PROGRAM PRG_ReadModbusSensorData
VAR
	
	CurrentReadTarget			: EN_ModbusReadTarget := EN_ModbusReadTarget.READ_TARGET_PH;
	
	ProcessValueRegister		: WORD := 2089;
	TemperatureRegister			: WORD := 2409;
	PhSensorUnitId				: BYTE := 1;
	OrpSensorUnitId				: BYTE := 2;
	RegQuantityToRead			: WORD :=10;
	
	currentUnitId				: BYTE := PhSensorUnitId;
	currentModbusRegister		: WORD := ProcessValueRegister;

	ModbusBusy					: BOOL := FALSE;

	(* diagnostics *)	
	LastModbusError				: ST_ModbusErrorDiagnostics;
	LastErrorstate				: INT;
	CurrentState				: INT;
	CounterError				: INT := 0;
	CounterSuccess				: INT := 0;
	
	firstCall					: BOOL := TRUE;	
	
	scaleFactorPh				: REAL :=   1.219512195; (* 0.980167935 *);  		
	offsetPh					: REAL := 	-1.280487805; (* -0.0216290391086993 *);	


	scaleFactorOrp				: REAL := 0.999321727334388;
	offsetOrp					: REAL := 0.0;			
	
END_VAR

(* looping through pH, pH-T, ORP, ORP-T reading the latest values *)
IF firstCall THEN
	PhModbus.ReadRegs( Execute := FALSE);
	OrpModbus.ReadRegs( Execute := FALSE);
	firstCall := FALSE;
END_IF	

CASE  CurrentReadTarget OF 
	EN_ModbusReadTarget.READ_TARGET_PH:
		PhModbus.Readregs (UnitID 		:= PhSensorUnitId ,
   							Quantity   	:= RegQuantityToRead,
   							MBAddr    	:= ProcessValueRegister,
   							cbLength    := RegQuantityToRead*2,
   							pMemoryAddr := ADR(PhValueArrayIn),   
   							Execute    	:= TRUE,
   							Timeout    	:= T#300MS,
							Busy 		=> ModbusBusy	
						  );
		
		IF NOT ModbusBusy THEN
			PhModbus.ReadRegs(Execute:= FALSE);
			CurrentReadTarget := EN_ModbusReadTarget.READ_TARGET_PH_T;
	
			IF PhModbus.Error THEN
				LastModbusError 	:= PhModbus.ErrorDiagnostics;
				LastErrorstate 		:= CurrentState;
				CounterError 		:= CounterError + 1;
				phLastReadingValid 	:= FALSE;
			ELSE
				CounterSuccess 		:= CounterSuccess + 1;
				phLastReadingValid 	:= TRUE;
				phCurrent			:= PhValueArrayIn[1]*scaleFactorPh + offsetPh;
			END_IF
		END_IF
		
	EN_ModbusReadTarget.READ_TARGET_PH_T:
		PhModbus.Readregs (UnitID 		:= PhSensorUnitId ,
   							Quantity   	:= RegQuantityToRead,
   							MBAddr    	:= TemperatureRegister,
   							cbLength    := RegQuantityToRead*2,
   							pMemoryAddr := ADR(TPhValueArrayIn),   
   							Execute    	:= TRUE,
   							Timeout    	:= T#300MS,
							Busy 		=> ModbusBusy	
						  );
		
		IF NOT ModbusBusy THEN
			PhModbus.ReadRegs(Execute:= FALSE);	
			CurrentReadTarget := EN_ModbusReadTarget.READ_TARGET_ORP;

			IF PhModbus.Error THEN
				LastModbusError 	:= PhModbus.ErrorDiagnostics;
				LastErrorstate 		:= CurrentState;
				CounterError 		:= CounterError + 1;
				tPhLastReadingValid := FALSE;
			ELSE
				CounterSuccess 		:= CounterSuccess + 1;
				tPhLastReadingValid := TRUE;
				tPhCurrent			:= TPhValueArrayIn[1];
			END_IF
		END_IF
	
	EN_ModbusReadTarget.READ_TARGET_ORP:
		OrpModbus.Readregs (UnitID 		:= OrpSensorUnitId ,
   							Quantity   	:= RegQuantityToRead,
   							MBAddr    	:= ProcessValueRegister,
   							cbLength    := RegQuantityToRead*2,
   							pMemoryAddr := ADR(OrpValueArrayIn),   
   							Execute    	:= TRUE,
   							Timeout    	:= T#300MS,
							Busy 		=> ModbusBusy	
						  );
		
		IF NOT ModbusBusy THEN
			OrpModbus.ReadRegs(Execute:= FALSE);	
			CurrentReadTarget := EN_ModbusReadTarget.READ_TARGET_ORP_T;

			IF OrpModbus.Error THEN
				LastModbusError 	:= OrpModbus.ErrorDiagnostics;
				LastErrorstate 		:= CurrentState;
				CounterError 		:= CounterError + 1;
				orpLastReadingValid := FALSE;
			ELSE
				CounterSuccess 		:= CounterSuccess + 1;
				orpLastReadingValid := TRUE;
				orpCurrent			:= OrpValueArrayIn[1]*scaleFactorOrp + offsetOrp;
			END_IF
		END_IF

	EN_ModbusReadTarget.READ_TARGET_ORP_T:

		OrpModbus.Readregs (UnitID 		:= OrpSensorUnitId ,
   							Quantity   	:= RegQuantityToRead,
   							MBAddr    	:= TemperatureRegister,
   							cbLength    := RegQuantityToRead*2,
   							pMemoryAddr := ADR(TOrpValueArrayIn),   
   							Execute    	:= TRUE,
   							Timeout    	:= T#300MS,
							Busy 		=> ModbusBusy	
						  );
		
		IF NOT ModbusBusy THEN
			OrpModbus.ReadRegs(Execute:= FALSE);	
			CurrentReadTarget := EN_ModbusReadTarget.READ_TARGET_PH;

			IF OrpModbus.Error THEN
				LastModbusError := OrpModbus.ErrorDiagnostics;
				LastErrorstate 	:= CurrentState;
				CounterError 	:= CounterError + 1;
				tOrpLastReadingValid := FALSE;
			ELSE
				CounterSuccess 	:= CounterSuccess + 1;
				tOrpLastReadingValid := TRUE;
				tOrpCurrent	:= TOrpValueArrayIn[1];
			END_IF
		END_IF
	
END_CASE
			
IF tPhLastReadingValid AND tOrpLastReadingValid THEN
	currentMeanTemp := (tPhCurrent + tOrpCurrent)/2.0;
	currentTempValid := TRUE;
ELSIF tPhLastReadingValid AND NOT tOrpLastReadingValid THEN
	currentMeanTemp := tPhCurrent;
	currentTempValid := TRUE;
ELSIF NOT tPhLastReadingValid AND tOrpLastReadingValid THEN
	currentMeanTemp := tOrpCurrent;
	currentTempValid := TRUE;
ELSE 
	(* no valid temperature signal !! signal to stop temperature control, if active *)
	currentTempValid := FALSE;
END_IF

END_PROGRAM

(* stored: Version 1.1.0.1, ProductVersion 3.1.4022.7
   POU PRG_ReadModbusSensorData: Id {70e2d931-711b-4294-8461-921be22fe8d2}, SpecialFunc None *)
